TYPE T_FOD_Cfg :
STRUCT
END_STRUCT
END_TYPE

(* stored: Version 1.1.0.1, ProductVersion 3.1.0.23
   DUT T_FOD_Cfg: Id {87075845-8a93-438f-a417-db5ca69fc26e} *)
